TYPE ST_PARAMETERS_HMI :
STRUCT
END_STRUCT
END_TYPE

(* stored: Version 1.1.0.1, ProductVersion 3.1.4022.11
   DUT ST_PARAMETERS_HMI: Id {255cd7c9-0edd-4941-8f45-6fe521f5236b} *)
